{attribute 'hide'}
FUNCTION_BLOCK Test_NotificationWithStringArg EXTENDS T_UnitTestBase
VAR
    Source  : T_Notification;
    Handler : T_NotificationHandler;

    ResultString : T_MaxString;
    Args         : I_StreamReader;
    IsRaised     : BOOL;
	Assertion : T_Assertion;
END_VAR

{attribute 'analysis' := '-33'} // inhibit unused variable warning
METHOD RunTest
VAR_OUTPUT
    TestCompleted : BOOL;
    TestFailed    : BOOL;
END_VAR
Handler.FB_init(bInitRetains := FALSE,
                bInCopyCode  := FALSE);

Source.ClearNotificationHandlers().AddNotificationHandler(Handler);
Source.Args.Init(81);

Source.Args.Clear().Add_STRING('Big long string passed to the notification handler for later use');
Source.Raise();

IF Handler.IsRaised() THEN
    Args         := Handler.Args;
    ResultString := Args.Read_STRING();
END_IF

TestFailed S= NOT Assertion.AssertEquals_STRING(Source    := TestName,
                             Expected     := 'Big long string passed to the notification handler for later use',
                              Actual       := ResultString,
                              VariableName := 'ResultString');

TestCompleted := TRUE;
END_METHOD

END_FUNCTION_BLOCK

(* stored: Version 1.1.0.1, ProductVersion 3.1.4024.12
   POU Test_NotificationWithStringArg: Id {e1171451-9ffb-40b1-b7d0-7319c599907b}, SpecialFunc None
   Method RunTest: Id {eb6cd482-2f7c-4752-8e5d-ca8001dd58a6} *)
